ABB RAPID module: Module2.mod

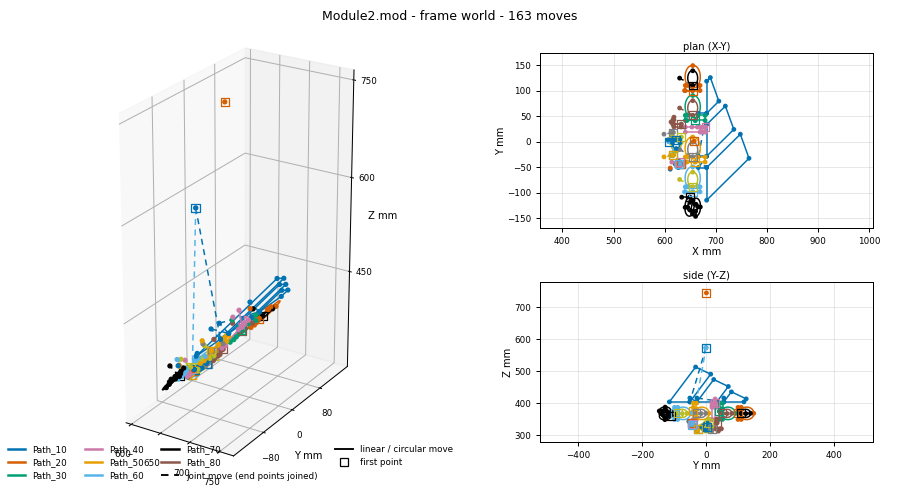
[picture p0: tool path of Module2.mod in frame world, 163 of 163 moves have a stored position in this frame; points joined in program order, loops and branches not executed]
MODULE Module1
    CONST robtarget Target_10:=[[150.037,154.697,5],[0.298836239,-0.640856382,-0.640856382,-0.298836239],[0,0,0,0],[9E+09,9E+09,9E+09,9E+09,9E+09,9E+09]];
    CONST robtarget Target_20:=[[86.037,154.697,5],[0.298836239,-0.640856382,-0.640856382,-0.298836239],[-1,0,-2,0],[9E+09,9E+09,9E+09,9E+09,9E+09,9E+09]];
    CONST robtarget Target_30:=[[168.037,17.697,5],[0.298836239,-0.640856382,-0.640856382,-0.298836239],[-1,0,-1,0],[9E+09,9E+09,9E+09,9E+09,9E+09,9E+09]];
    CONST robtarget Target_40:=[[215.231,45.775,5],[0.298836239,-0.640856382,-0.640856382,-0.298836239],[-1,0,-1,0],[9E+09,9E+09,9E+09,9E+09,9E+09,9E+09]];
    CONST robtarget Target_50:=[[150.037,154.697,5],[0.298836239,-0.640856382,-0.640856382,-0.298836239],[-1,0,-2,0],[9E+09,9E+09,9E+09,9E+09,9E+09,9E+09]];
    CONST robtarget Target_60:=[[172.037,154.697,5],[0.298836239,-0.640856382,-0.640856382,-0.298836239],[-1,0,-2,0],[9E+09,9E+09,9E+09,9E+09,9E+09,9E+09]];
    CONST robtarget Target_70:=[[224.668,66.765,5],[0.298836239,-0.640856382,-0.640856382,-0.298836239],[-1,0,-2,0],[9E+09,9E+09,9E+09,9E+09,9E+09,9E+09]];
    CONST robtarget Target_80:=[[270.264,94.172,5],[0.298836239,-0.640856382,-0.640856382,-0.298836239],[-1,0,-2,0],[9E+09,9E+09,9E+09,9E+09,9E+09,9E+09]];
    CONST robtarget Target_90:=[[234.037,154.697,5],[0.298836239,-0.640856382,-0.640856382,-0.298836239],[-1,0,-2,0],[9E+09,9E+09,9E+09,9E+09,9E+09,9E+09]];
    CONST robtarget Target_100:=[[172.037,154.697,5],[0.298836239,-0.640856382,-0.640856382,-0.298836239],[-1,0,-2,0],[9E+09,9E+09,9E+09,9E+09,9E+09,9E+09]];
    CONST robtarget Target_110:=[[256.037,154.697,5],[0.298836239,-0.640856382,-0.640856382,-0.298836239],[-1,0,-2,0],[9E+09,9E+09,9E+09,9E+09,9E+09,9E+09]];
    CONST robtarget Target_120:=[[279.922,115.116,5],[0.298836239,-0.640856382,-0.640856382,-0.298836239],[-1,0,-2,0],[9E+09,9E+09,9E+09,9E+09,9E+09,9E+09]];
    CONST robtarget Target_130:=[[326.037,142.697,5],[0.298836239,-0.640856382,-0.640856382,-0.298836239],[-1,1,-2,0],[9E+09,9E+09,9E+09,9E+09,9E+09,9E+09]];
    CONST robtarget Target_140:=[[319.037,154.697,5],[0.298836239,-0.640856382,-0.640856382,-0.298836239],[-1,1,-2,0],[9E+09,9E+09,9E+09,9E+09,9E+09,9E+09]];
    CONST robtarget Target_150:=[[256.037,154.697,5],[0.298836239,-0.640856382,-0.640856382,-0.298836239],[-1,0,-2,0],[9E+09,9E+09,9E+09,9E+09,9E+09,9E+09]];
    CONST robtarget Target_160:=[[300.621,199.726,5],[0.298836239,-0.640856382,-0.640856382,-0.298836239],[0,0,0,0],[9E+09,9E+09,9E+09,9E+09,9E+09,9E+09]];
    CONST robtarget Target_170:=[[300.621,175.964,5],[0.298836239,-0.640856382,-0.640856382,-0.298836239],[-1,0,-2,0],[9E+09,9E+09,9E+09,9E+09,9E+09,9E+09]];
    CONST robtarget Target_180:=[[310.571,175.964,5],[0.298836239,-0.640856382,-0.640856382,-0.298836239],[-1,1,-2,0],[9E+09,9E+09,9E+09,9E+09,9E+09,9E+09]];
    CONST robtarget Target_190:=[[310.571,182.87,5],[0.298836239,-0.640856382,-0.640856382,-0.298836239],[-1,1,-2,0],[9E+09,9E+09,9E+09,9E+09,9E+09,9E+09]];
    CONST robtarget Target_200:=[[327.056,175.147,5],[0.298836239,-0.640856382,-0.640856382,-0.298836239],[-1,1,-2,0],[9E+09,9E+09,9E+09,9E+09,9E+09,9E+09]];
    CONST robtarget Target_210:=[[349.482,199.504,5],[0.298836239,-0.640856382,-0.640856382,-0.298836239],[-1,1,-2,0],[9E+09,9E+09,9E+09,9E+09,9E+09,9E+09]];
    CONST robtarget Target_220:=[[327.205,224.231,5],[0.298836239,-0.640856382,-0.640856382,-0.298836239],[-1,1,-2,0],[9E+09,9E+09,9E+09,9E+09,9E+09,9E+09]];
    CONST robtarget Target_230:=[[310.571,216.434,5],[0.298836239,-0.640856382,-0.640856382,-0.298836239],[-1,1,-2,0],[9E+09,9E+09,9E+09,9E+09,9E+09,9E+09]];
    CONST robtarget Target_240:=[[310.571,223.489,5],[0.298836239,-0.640856382,-0.640856382,-0.298836239],[-1,1,-2,0],[9E+09,9E+09,9E+09,9E+09,9E+09,9E+09]];
    CONST robtarget Target_250:=[[300.621,223.489,5],[0.298836239,-0.640856382,-0.640856382,-0.298836239],[-1,1,-2,0],[9E+09,9E+09,9E+09,9E+09,9E+09,9E+09]];
    CONST robtarget Target_260:=[[300.621,199.726,5],[0.298836239,-0.640856382,-0.640856382,-0.298836239],[-1,1,-2,0],[9E+09,9E+09,9E+09,9E+09,9E+09,9E+09]];
    CONST robtarget Target_270:=[[242.106,191.558,5],[0.298836239,-0.640856382,-0.640856382,-0.298836239],[0,0,0,0],[9E+09,9E+09,9E+09,9E+09,9E+09,9E+09]];
    CONST robtarget Target_280:=[[242.106,159.627,5],[0.298836239,-0.640856382,-0.640856382,-0.298836239],[-1,0,-2,0],[9E+09,9E+09,9E+09,9E+09,9E+09,9E+09]];
    CONST robtarget Target_290:=[[252.056,159.627,5],[0.298836239,-0.640856382,-0.640856382,-0.298836239],[-1,0,-2,0],[9E+09,9E+09,9E+09,9E+09,9E+09,9E+09]];
    CONST robtarget Target_300:=[[252.056,182.573,5],[0.298836239,-0.640856382,-0.640856382,-0.298836239],[-1,0,-2,0],[9E+09,9E+09,9E+09,9E+09,9E+09,9E+09]];
    CONST robtarget Target_310:=[[268.467,175.147,5],[0.298836239,-0.640856382,-0.640856382,-0.298836239],[-1,0,-2,0],[9E+09,9E+09,9E+09,9E+09,9E+09,9E+09]];
    CONST robtarget Target_320:=[[290.967,199.504,5],[0.298836239,-0.640856382,-0.640856382,-0.298836239],[-1,0,-2,0],[9E+09,9E+09,9E+09,9E+09,9E+09,9E+09]];
    CONST robtarget Target_330:=[[268.542,224.231,5],[0.298836239,-0.640856382,-0.640856382,-0.298836239],[-1,0,-2,0],[9E+09,9E+09,9E+09,9E+09,9E+09,9E+09]];
    CONST robtarget Target_340:=[[252.056,216.36,5],[0.298836239,-0.640856382,-0.640856382,-0.298836239],[-1,0,-2,0],[9E+09,9E+09,9E+09,9E+09,9E+09,9E+09]];
    CONST robtarget Target_350:=[[252.056,223.489,5],[0.298836239,-0.640856382,-0.640856382,-0.298836239],[-1,0,-2,0],[9E+09,9E+09,9E+09,9E+09,9E+09,9E+09]];
    CONST robtarget Target_360:=[[242.106,223.489,5],[0.298836239,-0.640856382,-0.640856382,-0.298836239],[-1,0,-2,0],[9E+09,9E+09,9E+09,9E+09,9E+09,9E+09]];
    CONST robtarget Target_370:=[[242.106,191.558,5],[0.298836239,-0.640856382,-0.640856382,-0.298836239],[-1,0,-2,0],[9E+09,9E+09,9E+09,9E+09,9E+09,9E+09]];
    CONST robtarget Target_380:=[[229.126,158.35,5],[0.298836239,-0.640856382,-0.640856382,-0.298836239],[0,0,0,0],[9E+09,9E+09,9E+09,9E+09,9E+09,9E+09]];
    CONST robtarget Target_390:=[[229.126,168.33,5],[0.298836239,-0.640856382,-0.640856382,-0.298836239],[-1,0,-2,0],[9E+09,9E+09,9E+09,9E+09,9E+09,9E+09]];
    CONST robtarget Target_400:=[[219.146,168.33,5],[0.298836239,-0.640856382,-0.640856382,-0.298836239],[-1,0,-2,0],[9E+09,9E+09,9E+09,9E+09,9E+09,9E+09]];
    CONST robtarget Target_410:=[[219.146,158.35,5],[0.298836239,-0.640856382,-0.640856382,-0.298836239],[-1,0,-2,0],[9E+09,9E+09,9E+09,9E+09,9E+09,9E+09]];
    CONST robtarget Target_420:=[[229.126,158.35,5],[0.298836239,-0.640856382,-0.640856382,-0.298836239],[-1,0,-2,0],[9E+09,9E+09,9E+09,9E+09,9E+09,9E+09]];
    CONST robtarget Target_430:=[[229.185,175.964,5],[0.298836239,-0.640856382,-0.640856382,-0.298836239],[-1,0,-2,0],[9E+09,9E+09,9E+09,9E+09,9E+09,9E+09]];
    CONST robtarget Target_440:=[[229.185,223.489,5],[0.298836239,-0.640856382,-0.640856382,-0.298836239],[-1,0,-2,0],[9E+09,9E+09,9E+09,9E+09,9E+09,9E+09]];
    CONST robtarget Target_450:=[[219.309,223.489,5],[0.298836239,-0.640856382,-0.640856382,-0.298836239],[-1,0,-2,0],[9E+09,9E+09,9E+09,9E+09,9E+09,9E+09]];
    CONST robtarget Target_460:=[[219.309,175.964,5],[0.298836239,-0.640856382,-0.640856382,-0.298836239],[-1,0,-2,0],[9E+09,9E+09,9E+09,9E+09,9E+09,9E+09]];
    CONST robtarget Target_470:=[[229.185,175.964,5],[0.298836239,-0.640856382,-0.640856382,-0.298836239],[-1,0,-2,0],[9E+09,9E+09,9E+09,9E+09,9E+09,9E+09]];
    CONST robtarget Target_480:=[[160.794,191.558,5],[0.298836239,-0.640856382,-0.640856382,-0.298836239],[0,0,0,0],[9E+09,9E+09,9E+09,9E+09,9E+09,9E+09]];
    CONST robtarget Target_490:=[[160.794,159.627,5],[0.298836239,-0.640856382,-0.640856382,-0.298836239],[-1,0,-2,0],[9E+09,9E+09,9E+09,9E+09,9E+09,9E+09]];
    CONST robtarget Target_500:=[[170.745,159.627,5],[0.298836239,-0.640856382,-0.640856382,-0.298836239],[-1,0,-2,0],[9E+09,9E+09,9E+09,9E+09,9E+09,9E+09]];
    CONST robtarget Target_510:=[[170.745,182.573,5],[0.298836239,-0.640856382,-0.640856382,-0.298836239],[-1,0,-2,0],[9E+09,9E+09,9E+09,9E+09,9E+09,9E+09]];
    CONST robtarget Target_520:=[[187.155,175.147,5],[0.298836239,-0.640856382,-0.640856382,-0.298836239],[-1,0,-2,0],[9E+09,9E+09,9E+09,9E+09,9E+09,9E+09]];
    CONST robtarget Target_530:=[[209.655,199.504,5],[0.298836239,-0.640856382,-0.640856382,-0.298836239],[-1,0,-2,0],[9E+09,9E+09,9E+09,9E+09,9E+09,9E+09]];
    CONST robtarget Target_540:=[[187.23,224.231,5],[0.298836239,-0.640856382,-0.640856382,-0.298836239],[-1,0,-2,0],[9E+09,9E+09,9E+09,9E+09,9E+09,9E+09]];
    CONST robtarget Target_550:=[[170.745,216.36,5],[0.298836239,-0.640856382,-0.640856382,-0.298836239],[-1,0,-2,0],[9E+09,9E+09,9E+09,9E+09,9E+09,9E+09]];
    CONST robtarget Target_560:=[[170.745,223.489,5],[0.298836239,-0.640856382,-0.640856382,-0.298836239],[-1,0,-2,0],[9E+09,9E+09,9E+09,9E+09,9E+09,9E+09]];
    CONST robtarget Target_570:=[[160.794,223.489,5],[0.298836239,-0.640856382,-0.640856382,-0.298836239],[-1,0,-2,0],[9E+09,9E+09,9E+09,9E+09,9E+09,9E+09]];
    CONST robtarget Target_580:=[[160.794,191.558,5],[0.298836239,-0.640856382,-0.640856382,-0.298836239],[-1,0,-2,0],[9E+09,9E+09,9E+09,9E+09,9E+09,9E+09]];
    CONST robtarget Target_590:=[[102.279,199.726,5],[0.298836239,-0.640856382,-0.640856382,-0.298836239],[0,0,0,0],[9E+09,9E+09,9E+09,9E+09,9E+09,9E+09]];
    CONST robtarget Target_600:=[[102.279,175.964,5],[0.298836239,-0.640856382,-0.640856382,-0.298836239],[-1,0,-2,0],[9E+09,9E+09,9E+09,9E+09,9E+09,9E+09]];
    CONST robtarget Target_610:=[[112.23,175.964,5],[0.298836239,-0.640856382,-0.640856382,-0.298836239],[-1,0,-2,0],[9E+09,9E+09,9E+09,9E+09,9E+09,9E+09]];
    CONST robtarget Target_620:=[[112.23,182.87,5],[0.298836239,-0.640856382,-0.640856382,-0.298836239],[-1,0,-2,0],[9E+09,9E+09,9E+09,9E+09,9E+09,9E+09]];
    CONST robtarget Target_630:=[[128.715,175.147,5],[0.298836239,-0.640856382,-0.640856382,-0.298836239],[-1,0,-2,0],[9E+09,9E+09,9E+09,9E+09,9E+09,9E+09]];
    CONST robtarget Target_640:=[[151.141,199.504,5],[0.298836239,-0.640856382,-0.640856382,-0.298836239],[-1,0,-2,0],[9E+09,9E+09,9E+09,9E+09,9E+09,9E+09]];
    CONST robtarget Target_650:=[[128.863,224.231,5],[0.298836239,-0.640856382,-0.640856382,-0.298836239],[-1,0,-2,0],[9E+09,9E+09,9E+09,9E+09,9E+09,9E+09]];
    CONST robtarget Target_660:=[[112.23,216.434,5],[0.298836239,-0.640856382,-0.640856382,-0.298836239],[-1,0,-2,0],[9E+09,9E+09,9E+09,9E+09,9E+09,9E+09]];
    CONST robtarget Target_670:=[[112.23,223.489,5],[0.298836239,-0.640856382,-0.640856382,-0.298836239],[-1,0,-2,0],[9E+09,9E+09,9E+09,9E+09,9E+09,9E+09]];
    CONST robtarget Target_680:=[[102.279,223.489,5],[0.298836239,-0.640856382,-0.640856382,-0.298836239],[-1,0,-2,0],[9E+09,9E+09,9E+09,9E+09,9E+09,9E+09]];
    CONST robtarget Target_690:=[[102.279,199.726,5],[0.298836239,-0.640856382,-0.640856382,-0.298836239],[-1,0,-2,0],[9E+09,9E+09,9E+09,9E+09,9E+09,9E+09]];
    CONST robtarget Target_700:=[[91.957,208.934,5],[0.298836239,-0.640856382,-0.640856382,-0.298836239],[0,0,0,0],[9E+09,9E+09,9E+09,9E+09,9E+09,9E+09]];
    CONST robtarget Target_710:=[[86.138,219.85,5],[0.298836239,-0.640856382,-0.640856382,-0.298836239],[-1,0,-2,0],[9E+09,9E+09,9E+09,9E+09,9E+09,9E+09]];
    CONST robtarget Target_720:=[[72.056,224.231,5],[0.298836239,-0.640856382,-0.640856382,-0.298836239],[-1,0,-2,0],[9E+09,9E+09,9E+09,9E+09,9E+09,9E+09]];
    CONST robtarget Target_730:=[[58.848,220.314,5],[0.298836239,-0.640856382,-0.640856382,-0.298836239],[-1,0,-2,0],[9E+09,9E+09,9E+09,9E+09,9E+09,9E+09]];
    CONST robtarget Target_740:=[[58.996,200.432,5],[0.298836239,-0.640856382,-0.640856382,-0.298836239],[-1,0,-2,0],[9E+09,9E+09,9E+09,9E+09,9E+09,9E+09]];
    CONST robtarget Target_750:=[[78.303,193.127,5],[0.298836239,-0.640856382,-0.640856382,-0.298836239],[-1,0,-2,0],[9E+09,9E+09,9E+09,9E+09,9E+09,9E+09]];
    CONST robtarget Target_760:=[[81.264,188.811,5],[0.298836239,-0.640856382,-0.640856382,-0.298836239],[-1,0,-2,0],[9E+09,9E+09,9E+09,9E+09,9E+09,9E+09]];
    CONST robtarget Target_770:=[[73.245,183.464,5],[0.298836239,-0.640856382,-0.640856382,-0.298836239],[-1,0,-2,0],[9E+09,9E+09,9E+09,9E+09,9E+09,9E+09]];
    CONST robtarget Target_780:=[[66.896,185.358,5],[0.298836239,-0.640856382,-0.640856382,-0.298836239],[-1,0,-2,0],[9E+09,9E+09,9E+09,9E+09,9E+09,9E+09]];
    CONST robtarget Target_790:=[[64.334,190.444,5],[0.298836239,-0.640856382,-0.640856382,-0.298836239],[-1,0,-2,0],[9E+09,9E+09,9E+09,9E+09,9E+09,9E+09]];
    CONST robtarget Target_800:=[[54.457,190.444,5],[0.298836239,-0.640856382,-0.640856382,-0.298836239],[-1,0,-2,0],[9E+09,9E+09,9E+09,9E+09,9E+09,9E+09]];
    CONST robtarget Target_810:=[[59.804,179.269,5],[0.298836239,-0.640856382,-0.640856382,-0.298836239],[-1,0,-2,0],[9E+09,9E+09,9E+09,9E+09,9E+09,9E+09]];
    CONST robtarget Target_820:=[[72.873,175.147,5],[0.298836239,-0.640856382,-0.640856382,-0.298836239],[-1,0,-2,0],[9E+09,9E+09,9E+09,9E+09,9E+09,9E+09]];
    CONST robtarget Target_830:=[[86.193,179.12,5],[0.298836239,-0.640856382,-0.640856382,-0.298836239],[-1,0,-2,0],[9E+09,9E+09,9E+09,9E+09,9E+09,9E+09]];
    CONST robtarget Target_840:=[[86.008,198.854,5],[0.298836239,-0.640856382,-0.640856382,-0.298836239],[-1,0,-2,0],[9E+09,9E+09,9E+09,9E+09,9E+09,9E+09]];
    CONST robtarget Target_850:=[[66.079,206.298,5],[0.298836239,-0.640856382,-0.640856382,-0.298836239],[-1,0,-2,0],[9E+09,9E+09,9E+09,9E+09,9E+09,9E+09]];
    CONST robtarget Target_860:=[[65.819,214.392,5],[0.298836239,-0.640856382,-0.640856382,-0.298836239],[-1,0,-2,0],[9E+09,9E+09,9E+09,9E+09,9E+09,9E+09]];
    CONST robtarget Target_870:=[[72.279,215.989,5],[0.298836239,-0.640856382,-0.640856382,-0.298836239],[-1,0,-2,0],[9E+09,9E+09,9E+09,9E+09,9E+09,9E+09]];
    CONST robtarget Target_880:=[[78.851,213.947,5],[0.298836239,-0.640856382,-0.640856382,-0.298836239],[-1,0,-2,0],[9E+09,9E+09,9E+09,9E+09,9E+09,9E+09]];
    CONST robtarget Target_890:=[[81.784,208.934,5],[0.298836239,-0.640856382,-0.640856382,-0.298836239],[-1,0,-2,0],[9E+09,9E+09,9E+09,9E+09,9E+09,9E+09]];
    CONST robtarget Target_900:=[[91.957,208.934,5],[0.298836239,-0.640856382,-0.640856382,-0.298836239],[-1,0,-2,0],[9E+09,9E+09,9E+09,9E+09,9E+09,9E+09]];
    CONST robtarget Target_910:=[[234.809,236.833,5],[0.298836239,-0.640856382,-0.640856382,-0.298836239],[0,0,0,0],[9E+09,9E+09,9E+09,9E+09,9E+09,9E+09]];
    CONST robtarget Target_920:=[[234.809,260.29,5],[0.298836239,-0.640856382,-0.640856382,-0.298836239],[-1,0,-2,0],[9E+09,9E+09,9E+09,9E+09,9E+09,9E+09]];
    CONST robtarget Target_930:=[[239.033,264.958,5],[0.298836239,-0.640856382,-0.640856382,-0.298836239],[-1,0,-2,0],[9E+09,9E+09,9E+09,9E+09,9E+09,9E+09]];
    CONST robtarget Target_940:=[[243.218,260.29,5],[0.298836239,-0.640856382,-0.640856382,-0.298836239],[-1,0,-2,0],[9E+09,9E+09,9E+09,9E+09,9E+09,9E+09]];
    CONST robtarget Target_950:=[[248.609,260.29,5],[0.298836239,-0.640856382,-0.640856382,-0.298836239],[-1,0,-2,0],[9E+09,9E+09,9E+09,9E+09,9E+09,9E+09]];
    CONST robtarget Target_960:=[[245.974,267.15,5],[0.298836239,-0.640856382,-0.640856382,-0.298836239],[-1,0,-2,0],[9E+09,9E+09,9E+09,9E+09,9E+09,9E+09]];
    CONST robtarget Target_970:=[[239.033,269.665,5],[0.298836239,-0.640856382,-0.640856382,-0.298836239],[-1,0,-2,0],[9E+09,9E+09,9E+09,9E+09,9E+09,9E+09]];
    CONST robtarget Target_980:=[[232.073,267.15,5],[0.298836239,-0.640856382,-0.640856382,-0.298836239],[-1,0,-2,0],[9E+09,9E+09,9E+09,9E+09,9E+09,9E+09]];
    CONST robtarget Target_990:=[[229.417,260.29,5],[0.298836239,-0.640856382,-0.640856382,-0.298836239],[-1,0,-2,0],[9E+09,9E+09,9E+09,9E+09,9E+09,9E+09]];
    CONST robtarget Target_1000:=[[229.417,236.833,5],[0.298836239,-0.640856382,-0.640856382,-0.298836239],[-1,0,-2,0],[9E+09,9E+09,9E+09,9E+09,9E+09,9E+09]];
    CONST robtarget Target_1010:=[[234.809,236.833,5],[0.298836239,-0.640856382,-0.640856382,-0.298836239],[-1,0,-2,0],[9E+09,9E+09,9E+09,9E+09,9E+09,9E+09]];
    CONST robtarget Target_1020:=[[218.594,262.825,5],[0.298836239,-0.640856382,-0.640856382,-0.298836239],[0,0,0,0],[9E+09,9E+09,9E+09,9E+09,9E+09,9E+09]];
    CONST robtarget Target_1030:=[[222.014,266.245,5],[0.298836239,-0.640856382,-0.640856382,-0.298836239],[-1,0,-2,0],[9E+09,9E+09,9E+09,9E+09,9E+09,9E+09]];
    CONST robtarget Target_1040:=[[218.594,269.665,5],[0.298836239,-0.640856382,-0.640856382,-0.298836239],[-1,0,-2,0],[9E+09,9E+09,9E+09,9E+09,9E+09,9E+09]];
    CONST robtarget Target_1050:=[[215.254,266.245,5],[0.298836239,-0.640856382,-0.640856382,-0.298836239],[-1,0,-2,0],[9E+09,9E+09,9E+09,9E+09,9E+09,9E+09]];
    CONST robtarget Target_1060:=[[218.594,262.825,5],[0.298836239,-0.640856382,-0.640856382,-0.298836239],[-1,0,-2,0],[9E+09,9E+09,9E+09,9E+09,9E+09,9E+09]];
    CONST robtarget Target_1070:=[[209.501,236.833,5],[0.298836239,-0.640856382,-0.640856382,-0.298836239],[0,0,0,0],[9E+09,9E+09,9E+09,9E+09,9E+09,9E+09]];
    CONST robtarget Target_1080:=[[209.501,269.343,5],[0.298836239,-0.640856382,-0.640856382,-0.298836239],[-1,0,-2,0],[9E+09,9E+09,9E+09,9E+09,9E+09,9E+09]];
    CONST robtarget Target_1090:=[[198.879,269.343,5],[0.298836239,-0.640856382,-0.640856382,-0.298836239],[-1,0,-2,0],[9E+09,9E+09,9E+09,9E+09,9E+09,9E+09]];
    CONST robtarget Target_1100:=[[186.325,265.048,5],[0.298836239,-0.640856382,-0.640856382,-0.298836239],[-1,0,-2,0],[9E+09,9E+09,9E+09,9E+09,9E+09,9E+09]];
    CONST robtarget Target_1110:=[[181.618,253.209,5],[0.298836239,-0.640856382,-0.640856382,-0.298836239],[-1,0,-2,0],[9E+09,9E+09,9E+09,9E+09,9E+09,9E+09]];
    CONST robtarget Target_1120:=[[186.325,241.249,5],[0.298836239,-0.640856382,-0.640856382,-0.298836239],[-1,0,-2,0],[9E+09,9E+09,9E+09,9E+09,9E+09,9E+09]];
    CONST robtarget Target_1130:=[[198.879,236.833,5],[0.298836239,-0.640856382,-0.640856382,-0.298836239],[-1,0,-2,0],[9E+09,9E+09,9E+09,9E+09,9E+09,9E+09]];
    CONST robtarget Target_1140:=[[209.501,236.833,5],[0.298836239,-0.640856382,-0.640856382,-0.298836239],[-1,0,-2,0],[9E+09,9E+09,9E+09,9E+09,9E+09,9E+09]];
    CONST robtarget Target_1150:=[[156.471,236.391,5],[0.298836239,-0.640856382,-0.640856382,-0.298836239],[0,0,0,0],[9E+09,9E+09,9E+09,9E+09,9E+09,9E+09]];
    CONST robtarget Target_1160:=[[166.248,246.168,5],[0.298836239,-0.640856382,-0.640856382,-0.298836239],[-1,0,-2,0],[9E+09,9E+09,9E+09,9E+09,9E+09,9E+09]];
    CONST robtarget Target_1170:=[[156.471,255.905,5],[0.298836239,-0.640856382,-0.640856382,-0.298836239],[-1,0,-2,0],[9E+09,9E+09,9E+09,9E+09,9E+09,9E+09]];
    CONST robtarget Target_1180:=[[146.734,246.168,5],[0.298836239,-0.640856382,-0.640856382,-0.298836239],[-1,0,-2,0],[9E+09,9E+09,9E+09,9E+09,9E+09,9E+09]];
    CONST robtarget Target_1190:=[[156.471,236.391,5],[0.298836239,-0.640856382,-0.640856382,-0.298836239],[-1,0,-2,0],[9E+09,9E+09,9E+09,9E+09,9E+09,9E+09]];
    CONST robtarget Target_1200:=[[156.471,238.523,5],[0.298836239,-0.640856382,-0.640856382,-0.298836239],[0,0,0,0],[9E+09,9E+09,9E+09,9E+09,9E+09,9E+09]];
    CONST robtarget Target_1210:=[[163.914,246.168,5],[0.298836239,-0.640856382,-0.640856382,-0.298836239],[-1,0,-2,0],[9E+09,9E+09,9E+09,9E+09,9E+09,9E+09]];
    CONST robtarget Target_1220:=[[156.471,253.772,5],[0.298836239,-0.640856382,-0.640856382,-0.298836239],[-1,0,-2,0],[9E+09,9E+09,9E+09,9E+09,9E+09,9E+09]];
    CONST robtarget Target_1230:=[[149.027,246.168,5],[0.298836239,-0.640856382,-0.640856382,-0.298836239],[-1,0,-2,0],[9E+09,9E+09,9E+09,9E+09,9E+09,9E+09]];
    CONST robtarget Target_1240:=[[156.471,238.523,5],[0.298836239,-0.640856382,-0.640856382,-0.298836239],[-1,0,-2,0],[9E+09,9E+09,9E+09,9E+09,9E+09,9E+09]];
    CONST robtarget Target_1250:=[[174.174,262.825,5],[0.298836239,-0.640856382,-0.640856382,-0.298836239],[0,0,0,0],[9E+09,9E+09,9E+09,9E+09,9E+09,9E+09]];
    CONST robtarget Target_1260:=[[177.594,266.245,5],[0.298836239,-0.640856382,-0.640856382,-0.298836239],[-1,0,-2,0],[9E+09,9E+09,9E+09,9E+09,9E+09,9E+09]];
    CONST robtarget Target_1270:=[[174.174,269.665,5],[0.298836239,-0.640856382,-0.640856382,-0.298836239],[-1,0,-2,0],[9E+09,9E+09,9E+09,9E+09,9E+09,9E+09]];
    CONST robtarget Target_1280:=[[170.835,266.245,5],[0.298836239,-0.640856382,-0.640856382,-0.298836239],[-1,0,-2,0],[9E+09,9E+09,9E+09,9E+09,9E+09,9E+09]];
    CONST robtarget Target_1290:=[[174.174,262.825,5],[0.298836239,-0.640856382,-0.640856382,-0.298836239],[-1,0,-2,0],[9E+09,9E+09,9E+09,9E+09,9E+09,9E+09]];
    CONST robtarget Target_1300:=[[160.494,241.018,5],[0.298836239,-0.640856382,-0.640856382,-0.298836239],[0,0,0,0],[9E+09,9E+09,9E+09,9E+09,9E+09,9E+09]];
    CONST robtarget Target_1310:=[[160.494,251.076,5],[0.298836239,-0.640856382,-0.640856382,-0.298836239],[-1,0,-2,0],[9E+09,9E+09,9E+09,9E+09,9E+09,9E+09]];
    CONST robtarget Target_1320:=[[157.557,251.076,5],[0.298836239,-0.640856382,-0.640856382,-0.298836239],[-1,0,-2,0],[9E+09,9E+09,9E+09,9E+09,9E+09,9E+09]];
    CONST robtarget Target_1330:=[[157.557,247.576,5],[0.298836239,-0.640856382,-0.640856382,-0.298836239],[-1,0,-2,0],[9E+09,9E+09,9E+09,9E+09,9E+09,9E+09]];
    CONST robtarget Target_1340:=[[157.235,247.576,5],[0.298836239,-0.640856382,-0.640856382,-0.298836239],[-1,0,-2,0],[9E+09,9E+09,9E+09,9E+09,9E+09,9E+09]];
    CONST robtarget Target_1350:=[[155.143,251.076,5],[0.298836239,-0.640856382,-0.640856382,-0.298836239],[-1,0,-2,0],[9E+09,9E+09,9E+09,9E+09,9E+09,9E+09]];
    CONST robtarget Target_1360:=[[151.602,251.076,5],[0.298836239,-0.640856382,-0.640856382,-0.298836239],[-1,0,-2,0],[9E+09,9E+09,9E+09,9E+09,9E+09,9E+09]];
    CONST robtarget Target_1370:=[[154.097,247.214,5],[0.298836239,-0.640856382,-0.640856382,-0.298836239],[-1,0,-2,0],[9E+09,9E+09,9E+09,9E+09,9E+09,9E+09]];
    CONST robtarget Target_1380:=[[152.689,246.087,5],[0.298836239,-0.640856382,-0.640856382,-0.298836239],[-1,0,-2,0],[9E+09,9E+09,9E+09,9E+09,9E+09,9E+09]];
    CONST robtarget Target_1390:=[[152.166,244.277,5],[0.298836239,-0.640856382,-0.640856382,-0.298836239],[-1,0,-2,0],[9E+09,9E+09,9E+09,9E+09,9E+09,9E+09]];
    CONST robtarget Target_1400:=[[153.152,241.923,5],[0.298836239,-0.640856382,-0.640856382,-0.298836239],[-1,0,-2,0],[9E+09,9E+09,9E+09,9E+09,9E+09,9E+09]];
    CONST robtarget Target_1410:=[[155.787,241.018,5],[0.298836239,-0.640856382,-0.640856382,-0.298836239],[-1,0,-2,0],[9E+09,9E+09,9E+09,9E+09,9E+09,9E+09]];
    CONST robtarget Target_1420:=[[160.494,241.018,5],[0.298836239,-0.640856382,-0.640856382,-0.298836239],[-1,0,-2,0],[9E+09,9E+09,9E+09,9E+09,9E+09,9E+09]];
    CONST robtarget Target_55:=[[150.037,154.697,25],[0.298836239,-0.640856382,-0.640856382,-0.298836239],[-1,0,-2,0],[9E+09,9E+09,9E+09,9E+09,9E+09,9E+09]];
    CONST robtarget Target_105:=[[172.037,154.697,25],[0.298836239,-0.640856382,-0.640856382,-0.298836239],[-1,0,-2,0],[9E+09,9E+09,9E+09,9E+09,9E+09,9E+09]];
    CONST robtarget Target_155:=[[256.037,154.697,25],[0.298836239,-0.640856382,-0.640856382,-0.298836239],[-1,0,-2,0],[9E+09,9E+09,9E+09,9E+09,9E+09,9E+09]];
    CONST robtarget Target_265:=[[300.621,199.726,25],[0.298836239,-0.640856382,-0.640856382,-0.298836239],[-1,0,-2,0],[9E+09,9E+09,9E+09,9E+09,9E+09,9E+09]];
    CONST robtarget Target_375:=[[242.106,191.558,25],[0.298836239,-0.640856382,-0.640856382,-0.298836239],[-1,0,-2,0],[9E+09,9E+09,9E+09,9E+09,9E+09,9E+09]];
    CONST robtarget Target_425:=[[229.126,158.35,25],[0.298836239,-0.640856382,-0.640856382,-0.298836239],[-1,0,-2,0],[9E+09,9E+09,9E+09,9E+09,9E+09,9E+09]];
    CONST robtarget Target_475:=[[229.185,175.964,25],[0.298836239,-0.640856382,-0.640856382,-0.298836239],[-1,0,-2,0],[9E+09,9E+09,9E+09,9E+09,9E+09,9E+09]];
    CONST robtarget Target_585:=[[160.794,191.558,25],[0.298836239,-0.640856382,-0.640856382,-0.298836239],[-1,0,-2,0],[9E+09,9E+09,9E+09,9E+09,9E+09,9E+09]];
    CONST robtarget Target_695:=[[102.279,199.726,25],[0.298836239,-0.640856382,-0.640856382,-0.298836239],[-1,0,-2,0],[9E+09,9E+09,9E+09,9E+09,9E+09,9E+09]];
    CONST robtarget Target_905:=[[91.957,208.934,25],[0.298836239,-0.640856382,-0.640856382,-0.298836239],[-1,0,-2,0],[9E+09,9E+09,9E+09,9E+09,9E+09,9E+09]];
    CONST robtarget Target_1015:=[[234.809,236.833,25],[0.298836239,-0.640856382,-0.640856382,-0.298836239],[-1,0,-2,0],[9E+09,9E+09,9E+09,9E+09,9E+09,9E+09]];
    CONST robtarget Target_1055:=[[215.254,266.245,25],[0.298836239,-0.640856382,-0.640856382,-0.298836239],[-1,0,-2,0],[9E+09,9E+09,9E+09,9E+09,9E+09,9E+09]];
    CONST robtarget Target_1145:=[[209.501,236.833,25],[0.298836239,-0.640856382,-0.640856382,-0.298836239],[-1,0,-2,0],[9E+09,9E+09,9E+09,9E+09,9E+09,9E+09]];
    CONST robtarget Target_1185:=[[146.734,246.168,25],[0.298836239,-0.640856382,-0.640856382,-0.298836239],[-1,0,-2,0],[9E+09,9E+09,9E+09,9E+09,9E+09,9E+09]];
    CONST robtarget Target_1235:=[[149.027,246.168,25],[0.298836239,-0.640856382,-0.640856382,-0.298836239],[-1,0,-2,0],[9E+09,9E+09,9E+09,9E+09,9E+09,9E+09]];
    CONST robtarget Target_1285:=[[170.835,266.245,25],[0.298836239,-0.640856382,-0.640856382,-0.298836239],[-1,0,-2,0],[9E+09,9E+09,9E+09,9E+09,9E+09,9E+09]];
    CONST robtarget Target_1425:=[[160.494,241.018,25],[0.298836239,-0.640856382,-0.640856382,-0.298836239],[-1,0,-2,0],[9E+09,9E+09,9E+09,9E+09,9E+09,9E+09]];
    CONST robtarget Target_1430:=[[157.557,243.633,5],[0.298836239,-0.640856382,-0.640856382,-0.298836239],[0,0,0,0],[9E+09,9E+09,9E+09,9E+09,9E+09,9E+09]];
    CONST robtarget Target_1440:=[[157.557,245.162,5],[0.298836239,-0.640856382,-0.640856382,-0.298836239],[-1,0,-2,0],[9E+09,9E+09,9E+09,9E+09,9E+09,9E+09]];
    CONST robtarget Target_1450:=[[155.948,245.162,5],[0.298836239,-0.640856382,-0.640856382,-0.298836239],[-1,0,-2,0],[9E+09,9E+09,9E+09,9E+09,9E+09,9E+09]];
    CONST robtarget Target_1460:=[[155.063,244.357,5],[0.298836239,-0.640856382,-0.640856382,-0.298836239],[-1,0,-2,0],[9E+09,9E+09,9E+09,9E+09,9E+09,9E+09]];
    CONST robtarget Target_1470:=[[155.948,243.633,5],[0.298836239,-0.640856382,-0.640856382,-0.298836239],[-1,0,-2,0],[9E+09,9E+09,9E+09,9E+09,9E+09,9E+09]];
    CONST robtarget Target_1480:=[[157.557,243.633,5],[0.298836239,-0.640856382,-0.640856382,-0.298836239],[-1,0,-2,0],[9E+09,9E+09,9E+09,9E+09,9E+09,9E+09]];
    CONST robtarget Target_1785:=[[200.512085783,64.285097603,166.07719977],[0.23021145,-0.668582596,-0.668582596,-0.23021145],[0,-1,0,0],[9E+09,9E+09,9E+09,9E+09,9E+09,9E+09]];
    CONST robtarget Target_1490:=[[310.571,199.652,5],[0.298836239,-0.640856382,-0.640856382,-0.298836239],[0,0,0,0],[9E+09,9E+09,9E+09,9E+09,9E+09,9E+09]];
    CONST robtarget Target_1500:=[[324.977,183.687,5],[0.298836239,-0.640856382,-0.640856382,-0.298836239],[-1,1,-2,0],[9E+09,9E+09,9E+09,9E+09,9E+09,9E+09]];
    CONST robtarget Target_1510:=[[339.383,199.504,5],[0.298836239,-0.640856382,-0.640856382,-0.298836239],[-1,1,-2,0],[9E+09,9E+09,9E+09,9E+09,9E+09,9E+09]];
    CONST robtarget Target_1520:=[[324.977,215.692,5],[0.298836239,-0.640856382,-0.640856382,-0.298836239],[-1,1,-2,0],[9E+09,9E+09,9E+09,9E+09,9E+09,9E+09]];
    CONST robtarget Target_1530:=[[310.571,199.652,5],[0.298836239,-0.640856382,-0.640856382,-0.298836239],[-1,1,-2,0],[9E+09,9E+09,9E+09,9E+09,9E+09,9E+09]];
    CONST robtarget Target_1525:=[[324.977,215.692,25],[0.298836239,-0.640856382,-0.640856382,-0.298836239],[-1,0,-2,0],[9E+09,9E+09,9E+09,9E+09,9E+09,9E+09]];
    CONST robtarget Target_1540:=[[252.056,199.652,5],[0.298836239,-0.640856382,-0.640856382,-0.298836239],[-1,0,-2,0],[9E+09,9E+09,9E+09,9E+09,9E+09,9E+09]];
    CONST robtarget Target_1550:=[[266.462,183.687,5],[0.298836239,-0.640856382,-0.640856382,-0.298836239],[-1,0,-2,0],[9E+09,9E+09,9E+09,9E+09,9E+09,9E+09]];
    CONST robtarget Target_1560:=[[280.868,199.504,5],[0.298836239,-0.640856382,-0.640856382,-0.298836239],[-1,0,-2,0],[9E+09,9E+09,9E+09,9E+09,9E+09,9E+09]];
    CONST robtarget Target_1570:=[[266.462,215.692,5],[0.298836239,-0.640856382,-0.640856382,-0.298836239],[-1,0,-2,0],[9E+09,9E+09,9E+09,9E+09,9E+09,9E+09]];
    CONST robtarget Target_1580:=[[252.056,199.652,5],[0.298836239,-0.640856382,-0.640856382,-0.298836239],[0,0,0,0],[9E+09,9E+09,9E+09,9E+09,9E+09,9E+09]];
    CONST robtarget Target_1575:=[[266.462,215.692,25],[0.298836239,-0.640856382,-0.640856382,-0.298836239],[-1,0,-2,0],[9E+09,9E+09,9E+09,9E+09,9E+09,9E+09]];
    CONST robtarget Target_1590:=[[170.745,199.652,5],[0.298836239,-0.640856382,-0.640856382,-0.298836239],[-1,0,-2,0],[9E+09,9E+09,9E+09,9E+09,9E+09,9E+09]];
    CONST robtarget Target_1600:=[[185.151,183.687,5],[0.298836239,-0.640856382,-0.640856382,-0.298836239],[-1,0,-2,0],[9E+09,9E+09,9E+09,9E+09,9E+09,9E+09]];
    CONST robtarget Target_1610:=[[199.556,199.504,5],[0.298836239,-0.640856382,-0.640856382,-0.298836239],[-1,0,-2,0],[9E+09,9E+09,9E+09,9E+09,9E+09,9E+09]];
    CONST robtarget Target_1620:=[[185.151,215.692,5],[0.298836239,-0.640856382,-0.640856382,-0.298836239],[-1,0,-2,0],[9E+09,9E+09,9E+09,9E+09,9E+09,9E+09]];
    CONST robtarget Target_1630:=[[170.745,199.652,5],[0.298836239,-0.640856382,-0.640856382,-0.298836239],[0,0,0,0],[9E+09,9E+09,9E+09,9E+09,9E+09,9E+09]];
    CONST robtarget Target_1625:=[[185.151,215.692,25],[0.298836239,-0.640856382,-0.640856382,-0.298836239],[-1,0,-2,0],[9E+09,9E+09,9E+09,9E+09,9E+09,9E+09]];
    CONST robtarget Target_1640:=[[112.23,199.652,5],[0.298836239,-0.640856382,-0.640856382,-0.298836239],[-1,0,-2,0],[9E+09,9E+09,9E+09,9E+09,9E+09,9E+09]];
    CONST robtarget Target_1650:=[[126.636,183.687,5],[0.298836239,-0.640856382,-0.640856382,-0.298836239],[-1,0,-2,0],[9E+09,9E+09,9E+09,9E+09,9E+09,9E+09]];
    CONST robtarget Target_1660:=[[141.042,199.504,5],[0.298836239,-0.640856382,-0.640856382,-0.298836239],[-1,0,-2,0],[9E+09,9E+09,9E+09,9E+09,9E+09,9E+09]];
    CONST robtarget Target_1670:=[[126.636,215.692,5],[0.298836239,-0.640856382,-0.640856382,-0.298836239],[-1,0,-2,0],[9E+09,9E+09,9E+09,9E+09,9E+09,9E+09]];
    CONST robtarget Target_1680:=[[112.23,199.652,5],[0.298836239,-0.640856382,-0.640856382,-0.298836239],[0,0,0,0],[9E+09,9E+09,9E+09,9E+09,9E+09,9E+09]];
    CONST robtarget Target_1675:=[[126.636,215.692,25],[0.298836239,-0.640856382,-0.640856382,-0.298836239],[-1,0,-2,0],[9E+09,9E+09,9E+09,9E+09,9E+09,9E+09]];
    CONST robtarget Target_1690:=[[204.15,253.088,5],[0.298836239,-0.640856382,-0.640856382,-0.298836239],[-1,0,-2,0],[9E+09,9E+09,9E+09,9E+09,9E+09,9E+09]];
    CONST robtarget Target_1700:=[[204.15,264.998,5],[0.298836239,-0.640856382,-0.640856382,-0.298836239],[-1,0,-2,0],[9E+09,9E+09,9E+09,9E+09,9E+09,9E+09]];
    CONST robtarget Target_1710:=[[198.879,264.998,5],[0.298836239,-0.640856382,-0.640856382,-0.298836239],[-1,0,-2,0],[9E+09,9E+09,9E+09,9E+09,9E+09,9E+09]];
    CONST robtarget Target_1720:=[[190.128,261.92,5],[0.298836239,-0.640856382,-0.640856382,-0.298836239],[-1,0,-2,0],[9E+09,9E+09,9E+09,9E+09,9E+09,9E+09]];
    CONST robtarget Target_1730:=[[187.09,253.209,5],[0.298836239,-0.640856382,-0.640856382,-0.298836239],[-1,0,-2,0],[9E+09,9E+09,9E+09,9E+09,9E+09,9E+09]];
    CONST robtarget Target_1740:=[[190.128,244.377,5],[0.298836239,-0.640856382,-0.640856382,-0.298836239],[-1,0,-2,0],[9E+09,9E+09,9E+09,9E+09,9E+09,9E+09]];
    CONST robtarget Target_1750:=[[198.879,241.179,5],[0.298836239,-0.640856382,-0.640856382,-0.298836239],[-1,0,-2,0],[9E+09,9E+09,9E+09,9E+09,9E+09,9E+09]];
    CONST robtarget Target_1760:=[[204.15,241.179,5],[0.298836239,-0.640856382,-0.640856382,-0.298836239],[-1,0,-2,0],[9E+09,9E+09,9E+09,9E+09,9E+09,9E+09]];
    CONST robtarget Target_1770:=[[204.15,253.088,5],[0.298836239,-0.640856382,-0.640856382,-0.298836239],[0,0,0,0],[9E+09,9E+09,9E+09,9E+09,9E+09,9E+09]];
    CONST robtarget Target_1775:=[[204.15,253.088,25],[0.298836239,-0.640856382,-0.640856382,-0.298836239],[-1,0,-2,0],[9E+09,9E+09,9E+09,9E+09,9E+09,9E+09]];
    PERS tooldata MyNewTool:=[TRUE,[[40.305,0,141.61],[0.923879533,0,0.382683432,0]],[1,[0,0,1],[1,0,0,0],0,0,0]];
    TASK PERS wobjdata Workobject_test:=[FALSE,TRUE,"",[[803.749084033,-200.512,506.228906514],[0.633539788,-0.314049896,-0.314049896,0.633539788]],[[0,0,30],[1,0,0,0]]];
    CONST robtarget Target_1795:=[[220.663897892,-91.604542209,222.070073383],[0.298836239,-0.640856382,-0.640856382,-0.298836239],[0,0,0,1],[9E+09,9E+09,9E+09,9E+09,9E+09,9E+09]];
    CONST robtarget Target_1805:=[[201.762385931,-101.581232525,230.509595739],[0.084065498,0.709860066,0.696092568,-0.066983691],[-1,-1,0,1],[9E+09,9E+09,9E+09,9E+09,9E+09,9E+09]];
!***********************************************************
    !
    ! Module:  Module1
    !
    ! Description:
    !   <Insert description here>
    !
    ! Author: dsone
    !
    ! Version: 1.0
    !
    !***********************************************************


    !***********************************************************
    !
    ! Procedure main
    !
    !   This is the entry point of your program
    !
    !***********************************************************
    PROC main()
        !Add your code here
        SetDO DO_01,0;
        SetDO DO_02,1;
        WHILE TRUE DO
            IF DI_02=1 THEN
                SetDO DO_01,1;
                SetDO DO_02,0;
                Path_150;
                SetDO DO_01,0;
                SetDO DO_02,1;

            ELSEIF DI_01=1 THEN
                SetDO DO_01,1;
                SetDO DO_02,0;
                Path_10;
                Path_20;
                Path_25;
                Path_30;
                Path_35;
                Path_40;
                Path_50;
                Path_55;
                Path_60;
                Path_65;
                Path_70;
                Path_80;
                Path_90;
                Path_100;
                Path_102;
                Path_105;
                Path_110;
                Path_120;
                Path_130;
                Path_140;
                SetDO DO_01,0;
                SetDO DO_02,1;
            ENDIF
        ENDWHILE

    ENDPROC
    PROC Path_10()
        MoveJ Target_1785,v1000,z100,MyNewTool\WObj:=Workobject_test;
        MoveJ Target_10,v100,z0,MyNewTool\WObj:=Workobject_test;
        MoveL Target_20,v100,z0,MyNewTool\WObj:=Workobject_test;
        MoveL Target_30,v100,z0,MyNewTool\WObj:=Workobject_test;
        MoveL Target_40,v100,z0,MyNewTool\WObj:=Workobject_test;
        MoveL Target_50,v100,z0,MyNewTool\WObj:=Workobject_test;
        MoveJ Target_55,v100,z0,MyNewTool\WObj:=Workobject_test;
        MoveJ Target_60,v100,z0,MyNewTool\WObj:=Workobject_test;
        MoveL Target_70,v100,z0,MyNewTool\WObj:=Workobject_test;
        MoveL Target_80,v100,z0,MyNewTool\WObj:=Workobject_test;
        MoveL Target_90,v100,z0,MyNewTool\WObj:=Workobject_test;
        MoveL Target_100,v100,z0,MyNewTool\WObj:=Workobject_test;
        MoveJ Target_105,v100,z0,MyNewTool\WObj:=Workobject_test;
        MoveJ Target_110,v100,z0,MyNewTool\WObj:=Workobject_test;
        MoveL Target_120,v100,z0,MyNewTool\WObj:=Workobject_test;
        MoveL Target_130,v100,z0,MyNewTool\WObj:=Workobject_test;
        MoveL Target_140,v100,z0,MyNewTool\WObj:=Workobject_test;
        MoveL Target_150,v100,z0,MyNewTool\WObj:=Workobject_test;
        MoveJ Target_155,v1000,z100,MyNewTool\WObj:=Workobject_test;
    ENDPROC
    PROC Path_20()
        MoveJ Target_160,v100,z0,MyNewTool\WObj:=Workobject_test;
        MoveL Target_170,v100,z0,MyNewTool\WObj:=Workobject_test;
        MoveL Target_180,v100,z0,MyNewTool\WObj:=Workobject_test;
        MoveL Target_190,v100,z0,MyNewTool\WObj:=Workobject_test;
        MoveC Target_200,Target_210,v100,z0,MyNewTool\WObj:=Workobject_test;
        MoveC Target_220,Target_230,v100,z0,MyNewTool\WObj:=Workobject_test;
        MoveL Target_240,v100,z0,MyNewTool\WObj:=Workobject_test;
        MoveL Target_250,v100,z0,MyNewTool\WObj:=Workobject_test;
        MoveL Target_260,v100,z0,MyNewTool\WObj:=Workobject_test;
        MoveJ Target_265,v1000,z100,MyNewTool\WObj:=Workobject_test;
    ENDPROC
    PROC Path_30()
        MoveJ Target_270,v100,z0,MyNewTool\WObj:=Workobject_test;
        MoveL Target_280,v100,z0,MyNewTool\WObj:=Workobject_test;
        MoveL Target_290,v100,z0,MyNewTool\WObj:=Workobject_test;
        MoveL Target_300,v100,z0,MyNewTool\WObj:=Workobject_test;
        MoveC Target_310,Target_320,v100,z0,MyNewTool\WObj:=Workobject_test;
        MoveC Target_330,Target_340,v100,z0,MyNewTool\WObj:=Workobject_test;
        MoveL Target_350,v100,z0,MyNewTool\WObj:=Workobject_test;
        MoveL Target_360,v100,z0,MyNewTool\WObj:=Workobject_test;
        MoveL Target_370,v100,z0,MyNewTool\WObj:=Workobject_test;
        MoveJ Target_375,v1000,z100,MyNewTool\WObj:=Workobject_test;
    ENDPROC
    PROC Path_40()
        MoveJ Target_380,v100,z0,MyNewTool\WObj:=Workobject_test;
        MoveL Target_390,v100,z0,MyNewTool\WObj:=Workobject_test;
        MoveL Target_400,v100,z0,MyNewTool\WObj:=Workobject_test;
        MoveL Target_410,v100,z0,MyNewTool\WObj:=Workobject_test;
        MoveL Target_420,v100,z0,MyNewTool\WObj:=Workobject_test;
        MoveJ Target_425,v1000,z100,MyNewTool\WObj:=Workobject_test;
        MoveL Target_430,v100,z0,MyNewTool\WObj:=Workobject_test;
        MoveL Target_440,v100,z0,MyNewTool\WObj:=Workobject_test;
        MoveL Target_450,v100,z0,MyNewTool\WObj:=Workobject_test;
        MoveL Target_460,v100,z0,MyNewTool\WObj:=Workobject_test;
        MoveL Target_470,v100,z0,MyNewTool\WObj:=Workobject_test;
        MoveJ Target_475,v1000,z100,MyNewTool\WObj:=Workobject_test;
    ENDPROC
    PROC Path_50()
        MoveJ Target_480,v100,z0,MyNewTool\WObj:=Workobject_test;
        MoveL Target_490,v100,z0,MyNewTool\WObj:=Workobject_test;
        MoveL Target_500,v100,z0,MyNewTool\WObj:=Workobject_test;
        MoveL Target_510,v100,z0,MyNewTool\WObj:=Workobject_test;
        MoveC Target_520,Target_530,v100,z0,MyNewTool\WObj:=Workobject_test;
        MoveC Target_540,Target_550,v100,z0,MyNewTool\WObj:=Workobject_test;
        MoveL Target_560,v100,z0,MyNewTool\WObj:=Workobject_test;
        MoveL Target_570,v100,z0,MyNewTool\WObj:=Workobject_test;
        MoveL Target_580,v100,z0,MyNewTool\WObj:=Workobject_test;
        MoveJ Target_585,v1000,z100,MyNewTool\WObj:=Workobject_test;
    ENDPROC
    PROC Path_60()
        MoveJ Target_590,v100,z0,MyNewTool\WObj:=Workobject_test;
        MoveL Target_600,v100,z0,MyNewTool\WObj:=Workobject_test;
        MoveL Target_610,v100,z0,MyNewTool\WObj:=Workobject_test;
        MoveL Target_620,v100,z0,MyNewTool\WObj:=Workobject_test;
        MoveC Target_630,Target_640,v100,z0,MyNewTool\WObj:=Workobject_test;
        MoveC Target_650,Target_660,v100,z0,MyNewTool\WObj:=Workobject_test;
        MoveL Target_670,v100,z0,MyNewTool\WObj:=Workobject_test;
        MoveL Target_680,v100,z0,MyNewTool\WObj:=Workobject_test;
        MoveL Target_690,v100,z0,MyNewTool\WObj:=Workobject_test;
        MoveJ Target_695,v1000,z100,MyNewTool\WObj:=Workobject_test;
    ENDPROC
    PROC Path_70()
        MoveJ Target_700,v100,z0,MyNewTool\WObj:=Workobject_test;
        MoveC Target_710,Target_720,v100,z0,MyNewTool\WObj:=Workobject_test;
        MoveC Target_730,Target_740,v100,z0,MyNewTool\WObj:=Workobject_test;
        MoveL Target_750,v100,z0,MyNewTool\WObj:=Workobject_test;
        MoveC Target_760,Target_770,v100,z0,MyNewTool\WObj:=Workobject_test;
        MoveC Target_780,Target_790,v100,z0,MyNewTool\WObj:=Workobject_test;
        MoveL Target_800,v100,z0,MyNewTool\WObj:=Workobject_test;
        MoveC Target_810,Target_820,v100,z0,MyNewTool\WObj:=Workobject_test;
        MoveC Target_830,Target_840,v100,z0,MyNewTool\WObj:=Workobject_test;
        MoveL Target_850,v100,z0,MyNewTool\WObj:=Workobject_test;
        MoveC Target_860,Target_870,v100,z0,MyNewTool\WObj:=Workobject_test;
        MoveC Target_880,Target_890,v100,z0,MyNewTool\WObj:=Workobject_test;
        MoveL Target_900,v100,z0,MyNewTool\WObj:=Workobject_test;
        MoveJ Target_905,v1000,z100,MyNewTool\WObj:=Workobject_test;
    ENDPROC
    PROC Path_80()
        MoveJ Target_910,v100,z0,MyNewTool\WObj:=Workobject_test;
        MoveL Target_920,v100,z0,MyNewTool\WObj:=Workobject_test;
        MoveC Target_930,Target_940,v100,z0,MyNewTool\WObj:=Workobject_test;
        MoveL Target_950,v100,z0,MyNewTool\WObj:=Workobject_test;
        MoveC Target_960,Target_970,v100,z0,MyNewTool\WObj:=Workobject_test;
        MoveC Target_980,Target_990,v100,z0,MyNewTool\WObj:=Workobject_test;
        MoveL Target_1000,v100,z0,MyNewTool\WObj:=Workobject_test;
        MoveL Target_1010,v100,z0,MyNewTool\WObj:=Workobject_test;
        MoveJ Target_1015,v1000,z100,MyNewTool\WObj:=Workobject_test;
    ENDPROC
    PROC Path_90()
        MoveJ Target_1020,v100,z0,MyNewTool\WObj:=Workobject_test;
        MoveC Target_1030,Target_1040,v100,z0,MyNewTool\WObj:=Workobject_test;
        MoveC Target_1050,Target_1060,v100,z0,MyNewTool\WObj:=Workobject_test;
        MoveJ Target_1055,v1000,z100,MyNewTool\WObj:=Workobject_test;
    ENDPROC
    PROC Path_100()
        MoveJ Target_1070,v100,z0,MyNewTool\WObj:=Workobject_test;
        MoveL Target_1080,v100,z0,MyNewTool\WObj:=Workobject_test;
        MoveL Target_1090,v100,z0,MyNewTool\WObj:=Workobject_test;
        MoveC Target_1100,Target_1110,v100,z0,MyNewTool\WObj:=Workobject_test;
        MoveC Target_1120,Target_1130,v100,z0,MyNewTool\WObj:=Workobject_test;
        MoveL Target_1140,v100,z0,MyNewTool\WObj:=Workobject_test;
        MoveJ Target_1145,v1000,z100,MyNewTool\WObj:=Workobject_test;
    ENDPROC
    PROC Path_110()
        MoveJ Target_1150,v100,z0,MyNewTool\WObj:=Workobject_test;
        MoveC Target_1160,Target_1170,v100,z0,MyNewTool\WObj:=Workobject_test;
        MoveC Target_1180,Target_1190,v100,z0,MyNewTool\WObj:=Workobject_test;
        MoveJ Target_1185,v1000,z100,MyNewTool\WObj:=Workobject_test;
    ENDPROC
    PROC Path_120()
        MoveJ Target_1200,v100,z0,MyNewTool\WObj:=Workobject_test;
        MoveC Target_1210,Target_1220,v100,z0,MyNewTool\WObj:=Workobject_test;
        MoveC Target_1230,Target_1240,v100,z0,MyNewTool\WObj:=Workobject_test;
        MoveJ Target_1235,v1000,z100,MyNewTool\WObj:=Workobject_test;
    ENDPROC
    PROC Path_95()
        MoveL Target_1250,v100,z0,MyNewTool\WObj:=Workobject_test;
        MoveC Target_1260,Target_1270,v100,z0,MyNewTool\WObj:=Workobject_test;
        MoveC Target_1280,Target_1290,v100,z0,MyNewTool\WObj:=Workobject_test;
    ENDPROC
    PROC Path_130()
        MoveJ Target_1300,v100,z0,MyNewTool\WObj:=Workobject_test;
        MoveL Target_1310,v100,z0,MyNewTool\WObj:=Workobject_test;
        MoveL Target_1320,v100,z0,MyNewTool\WObj:=Workobject_test;
        MoveL Target_1330,v100,z0,MyNewTool\WObj:=Workobject_test;
        MoveL Target_1340,v100,z0,MyNewTool\WObj:=Workobject_test;
        MoveL Target_1350,v100,z0,MyNewTool\WObj:=Workobject_test;
        MoveL Target_1360,v100,z0,MyNewTool\WObj:=Workobject_test;
        MoveL Target_1370,v100,z0,MyNewTool\WObj:=Workobject_test;
        MoveC Target_1380,Target_1390,v100,z0,MyNewTool\WObj:=Workobject_test;
        MoveC Target_1400,Target_1410,v100,z0,MyNewTool\WObj:=Workobject_test;
        MoveL Target_1420,v100,z0,MyNewTool\WObj:=Workobject_test;
        MoveJ Target_1425,v1000,z100,MyNewTool\WObj:=Workobject_test;
    ENDPROC
    PROC Path_105()
        MoveJ Target_1250,v100,z0,MyNewTool\WObj:=Workobject_test;
        MoveC Target_1260,Target_1270,v100,z0,MyNewTool\WObj:=Workobject_test;
        MoveC Target_1280,Target_1290,v100,z0,MyNewTool\WObj:=Workobject_test;
        MoveJ Target_1285,v1000,z100,MyNewTool\WObj:=Workobject_test;
    ENDPROC
    PROC Path_140()
        MoveJ Target_1430,v100,z0,MyNewTool\WObj:=Workobject_test;
        MoveL Target_1440,v100,z0,MyNewTool\WObj:=Workobject_test;
        MoveL Target_1450,v100,z0,MyNewTool\WObj:=Workobject_test;
        MoveC Target_1460,Target_1470,v100,z0,MyNewTool\WObj:=Workobject_test;
        MoveL Target_1480,v100,z0,MyNewTool\WObj:=Workobject_test;
        MoveJ Target_1785,v1000,z100,MyNewTool\WObj:=Workobject_test;
    ENDPROC
    PROC Path_25()
        MoveJ Target_1490,v100,z0,MyNewTool\WObj:=Workobject_test;
        MoveC Target_1500,Target_1510,v100,z0,MyNewTool\WObj:=Workobject_test;
        MoveC Target_1520,Target_1530,v100,z0,MyNewTool\WObj:=Workobject_test;
        MoveJ Target_1525,v1000,z100,MyNewTool\WObj:=Workobject_test;
    ENDPROC
    PROC Path_35()
        MoveJ Target_1540,v100,z0,MyNewTool\WObj:=Workobject_test;
        MoveC Target_1550,Target_1560,v100,z0,MyNewTool\WObj:=Workobject_test;
        MoveC Target_1570,Target_1580,v100,z0,MyNewTool\WObj:=Workobject_test;
        MoveJ Target_1575,v1000,z100,MyNewTool\WObj:=Workobject_test;
    ENDPROC
    PROC Path_55()
        MoveJ Target_1590,v100,z0,MyNewTool\WObj:=Workobject_test;
        MoveC Target_1600,Target_1610,v100,z0,MyNewTool\WObj:=Workobject_test;
        MoveC Target_1620,Target_1630,v100,z0,MyNewTool\WObj:=Workobject_test;
        MoveJ Target_1625,v1000,z100,MyNewTool\WObj:=Workobject_test;
    ENDPROC
    PROC Path_65()
        MoveJ Target_1640,v100,z0,MyNewTool\WObj:=Workobject_test;
        MoveC Target_1650,Target_1660,v100,z0,MyNewTool\WObj:=Workobject_test;
        MoveC Target_1670,Target_1680,v100,z0,MyNewTool\WObj:=Workobject_test;
        MoveJ Target_1675,v1000,z100,MyNewTool\WObj:=Workobject_test;
    ENDPROC
    PROC Path_102()
        MoveJ Target_1690,v100,z0,MyNewTool\WObj:=Workobject_test;
        MoveL Target_1700,v100,z0,MyNewTool\WObj:=Workobject_test;
        MoveL Target_1710,v100,z0,MyNewTool\WObj:=Workobject_test;
        MoveC Target_1720,Target_1730,v100,z0,MyNewTool\WObj:=Workobject_test;
        MoveC Target_1740,Target_1750,v100,z0,MyNewTool\WObj:=Workobject_test;
        MoveL Target_1760,v100,z0,MyNewTool\WObj:=Workobject_test;
        MoveL Target_1770,v100,z0,MyNewTool\WObj:=Workobject_test;
        MoveJ Target_1775,v1000,z100,MyNewTool\WObj:=Workobject_test;
    ENDPROC
    PROC Path_150()
        MoveJ Target_1805,v1000,z0,MyNewTool\WObj:=Workobject_test;
    ENDPROC
ENDMODULE
